VAR_GLOBAL
    // Semantic version in machine-readable format.
    // Update it and commit it immediatly before setting a tag
    nVersionMajor: UINT := 2; // Major Version
    nVersionMinor: UINT := 10; // Minor Version
    nVersionPatch: UINT := 0; // Patch level

    //Structure arrays for the axes
    astAxes: ARRAY [1..GVL_APP.nAXIS_NUM] OF ST_AxisStruct; //Array of ST_AxisStruct for holding axis parameters and controls
    astPneumaticAxes: ARRAY [1..GVL_APP.nPNEUMATIC_AXIS_NUM] OF ST_PneumaticAxisStruct; //Array of ST_PneumaticAxisStruct for holding pneumatic axis parameters and controls
    afbPressureGroup: ARRAY[E_PneumaticAxisGroup.ePneumaticAxisGroup1..E_PneumaticAxisGroup.ePneumaticAxisGroup2] OF FB_PressureGroup;
    iAxis: UINT; //Index for for loops while going through axes
    iPneumaticAxis: UINT; //Index for for loops while going through pneumatic axes
    fbGetCurTaskIndex: GETCURTASKINDEX;
    bLocalMode: BOOL;
END_VAR

VAR_GLOBAL CONSTANT
    nMAX_AXIS_NAME: UINT := 32;
END_VAR

VAR_GLOBAL PERSISTENT
    astAxesPersistent: ARRAY [1..GVL_APP.nAXIS_NUM] OF ST_AxisPersistent;
    dtAtShutdownPersistent: DT; //Date and time when the CPU was powered off
END_VAR

(* stored: Version 1.1.0.1
   GVL GVL: Id {6a1837cf-595e-0fbe-2836-4fcfdeeb3666} *)
